// TIA Portal project "Labtest1" (V17)

(* hardware
DEVICE "S7-1200 station_1"  S7-1200 Station
   slot 0: "Rack_0"  S7-1200 Rack  Rack  V1.0
   slot 1: "PLC_1"  CPU 1214C DC/DC/DC  6ES7 214-1AG40-0XB0  V4.1
DEVICE "HMI_1"  KTP700 Basic PN
   slot 0: "HMI_1"  KTP700 Basic PN  6AV2 123-2GB03-0AX0  15.1.0.0
   slot 1: "HMI_RT_1"  KTP700 Basic PN  6AV2 123-2GB03-0AX0  15.1.0.0
   slot 5: "HMI_1.IE_CP_1"  PROFINET Interface  15.0.1.0
      slot 1: "PROFINET Interface_1"  PROFINET Interface
         slot 1: "Port_1"  Port
*)

// ===== PLC "PLC_1"  CPU 1214C DC/DC/DC =====

VAR_GLOBAL   // PLC tag table "Default tag table"
   "Analog_Input" AT %IW64 : Int;
   "Analog_Output" AT %Q0.0 : Bool;
   "EmptyTank" AT %I0.0 : Bool;
   "FilledTank" AT %I0.1 : Bool;
   "LED Indicator" AT %Q0.1 : Bool;
END_VAR

ORGANIZATION_BLOCK "Main"   // OB1, LAD, ProgramCycle
TITLE = "Main Program Sweep (Cycle)"
{ S7_Optimized_Access := 'TRUE' }
VERSION : 0.1
   VAR_INPUT
      Initial_Call : Bool;   // Initial call of this OB
      Remanence : Bool;   // =True, if remanent data are available
   END_VAR
BEGIN
END_ORGANIZATION_BLOCK

(* ===== HMI "HMI_RT_1" =====
connection "HMI_Connection_1": ETHERNET, SMART_S7_1200_OMS
*)